(* PLC project LadderSidePinFixture, greenforge-labs codescribe-fixture 1 *)
(* stored: creationDateTime 2020-01-01T00:00:00 *)

PROGRAM LD_SIDE_PIN
  VAR
    xSet : BOOL;
    xClear : BOOL;
    xCount : BOOL;
    xDone : BOOL;
    latch : SR;
    ctr : CTU;
  END_VAR

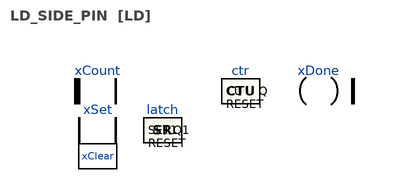
(* LD diagram, written out as Structured Text *)
latch(SET1 := xSet, RESET := xClear);
ctr(CU := xCount, RESET := latch.Q1);
xDone := ctr.Q;
END_PROGRAM
